(* IEC 61131-3 sources: CodesysTest/alpha/export/FBs, 6 files *)

(* ---- FB_CylinderLeak.pou.st ---- *)
(*#-#-#-#-#-#-#-#-#-#---Declaration---#-#-#-#-#-#-#-#-#-#-#-#-#*)

FUNCTION_BLOCK FB_CylinderLeak EXTENDS FB_PredictiveMaint
VAR_INPUT
	iExtended : BOOL;
	iRetracted : BOOL;
	maximumStrokeTime : REAL;
END_VAR
VAR_OUTPUT
	strokeTime : REAL;
END_VAR
VAR
	strokeTimer : TON := (PT := T#1H);
	extendedONS : R_TRIG;
	retractedONS : R_TRIG;
END_VAR
(*#-#-#-#-#-#-#-#-#-#---Implementation---#-#-#-#-#-#-#-#-#-#-#-#-#*)

extendedONS(CLK := iExtended);
retractedONS(CLK := iRetracted);

IF extendedONS.Q OR retractedONS.Q THEN
	strokeTime := TO_REAL(strokeTimer.ET) / 1000;
END_IF

strokeTimer(IN := NOT iExtended AND NOT iRetracted);

(* ---- FB_DriveTemp.pou.st ---- *)
(*#-#-#-#-#-#-#-#-#-#---Declaration---#-#-#-#-#-#-#-#-#-#-#-#-#*)

FUNCTION_BLOCK FB_DriveTemp EXTENDS FB_PredictiveMaint
VAR_INPUT
	iDriveTemp : DINT;
	maxTemp : REAL;
END_VAR
VAR_OUTPUT
	DriveTemp : REAL;
END_VAR
VAR
END_VAR
(*#-#-#-#-#-#-#-#-#-#---Implementation---#-#-#-#-#-#-#-#-#-#-#-#-#*)

DriveTemp := TO_REAL(iDriveTemp) / 10.0;

(* ---- FB_Throughput.pou.st ---- *)
(*#-#-#-#-#-#-#-#-#-#---Declaration---#-#-#-#-#-#-#-#-#-#-#-#-#*)

FUNCTION_BLOCK FB_Throughput
VAR_INPUT
	inCycle : BOOL;
	runtimeTimeout : REAL := 5.0;
	reset : BOOL;
END_VAR
VAR_OUTPUT
	BPM : REAL;
	BPMCycles : UDINT;
	BPMSeconds : UDINT;
	BPMIndication : STRING;
END_VAR
VAR
	resetRuntime : BOOL;
	resetRuntimeTimer : TON := (PT := T#0S);
	runtimeTimeoutTimer : Standard.TON;
	runtimeTimer : Standard.TON;
	actualRuntimeTimer : Standard.TON;
	timeoutONS : FB_ONS;
	inCycleONS : FB_ONS;
	runtimeSeconds : UDINT;
	runtimeMinutes : UDINT;
	runtimeHours : UDINT;
	runtimeDays : UDINT;
	runtimeSubtractedToGetFiveSeconds : UDINT;
	cycleStarted : BOOL;
	totalTempH : UDINT;
	totalTempM : UDINT;
	totalTempS : UDINT;
END_VAR
(*#-#-#-#-#-#-#-#-#-#---Implementation---#-#-#-#-#-#-#-#-#-#-#-#-#*)

// Runtime calculation. The goal is to capture actual runtime of the machine (i.e being used, including loading time)
inCycleONS(CLK := inCycle);
// Reset timeout time
IF inCycleONS.OSR THEN
	resetRuntime := TRUE;
	cycleStarted := TRUE;
	BPMCycles := BPMCycles + 1;
END_IF;

// After timeout, assume machine in unmanned
runtimeTimeoutTimer(IN := NOT resetRuntime, PT := TO_TIME(runtimeTimeout * 1000.0));
resetRuntime := FALSE;
timeoutONS(CLK := runtimeTimeoutTimer.Q);

// 1 second ticker while being used.
actualRuntimeTimer(IN := cycleStarted AND NOT actualRuntimeTimer.Q AND NOT runtimeTimeoutTimer.Q, PT := T#1S);

IF actualRuntimeTimer.Q THEN
	BPMSeconds := BPMSeconds + 1;
END_IF;

// Subtract 5 seconds after machine is abandoned
runtimeSubtractedToGetFiveSeconds := ANY_TO_UDINT(ABS(5.0 - runtimeTimeout));

IF timeoutONS.OSR THEN
	IF BPMSeconds > runtimeSubtractedToGetFiveSeconds THEN
		BPMSeconds := BPMSeconds - runtimeSubtractedToGetFiveSeconds;
	END_IF;
	cycleStarted := FALSE;
END_IF;

IF reset THEN
	BPMSeconds := 0;
	BPMCycles := 0;
END_IF;

// Concat to string for display
runtimeHours := BPMSeconds / 3600;
runtimeMinutes := (BPMSeconds MOD 3600) / 60;
runtimeSeconds := BPMSeconds MOD 60;

IF BPMSeconds <> 0 THEN
	BPM := ANY_TO_REAL(BPMCycles) / (ANY_TO_REAL(BPMSeconds) / 60.0);
ELSE
	BPM := 0.0;
END_IF;
BPMIndication := '';
BPMIndication := ANY_TO_STRING(runtimeHours);
BPMIndication := INSERT(BPMIndication, 'H  ', LEN(BPMIndication) + 2);
BPMIndication := INSERT(BPMIndication, ANY_TO_STRING(runtimeMinutes), LEN(BPMIndication));
BPMIndication := INSERT(BPMIndication, 'M ', LEN(BPMIndication));
BPMIndication := INSERT(BPMIndication, ANY_TO_STRING(runtimeSeconds), LEN(BPMIndication));
BPMIndication := INSERT(BPMIndication, 'S', LEN(BPMIndication));

(* ---- FB_WriteToFile.pou.st ---- *)
(*#-#-#-#-#-#-#-#-#-#---Declaration---#-#-#-#-#-#-#-#-#-#-#-#-#*)

FUNCTION_BLOCK FB_WriteToFile
VAR_INPUT
   xFilePath: STRING;
   xText_Write: STRING(5000);
   xAppend_OverWrite: BOOL;
   xAppend_Pos: UDINT;
   xWrite: BOOL;
   xRead: BOOL;
   xLine_No_To_Read: UDINT;
END_VAR
VAR_OUTPUT
   xText_Read: STRING(5000);
   xDone: BOOL;
END_VAR
VAR

// Write Variables
   xWrite_Trig: R_TRIG;
   xStart_Write: BOOL;
   xNew_Line: STRING(5000);

// Read Variables
   xRead_Trig: R_TRIG;
   xStart_Read: BOOL;
   xLine_Read: UDINT;

   hFile           : SysFile.RTS_IEC_HANDLE := SysFile.HandleConstants.RTS_INVALID_HANDLE;
   udiBytesRead    : LWORD;
   udiBytesCopied   : UDINT;
   udiWrite      : LWORD;
   udiFileSize     : UDINT;
   udiPos         : UDINT;

//(* Error Codes *)
   udiPosError          : SysFile.RTS_IEC_RESULT;
   udiCopyError      : SysFile.RTS_IEC_RESULT;
   udiDeleteError1      : SysFile.RTS_IEC_RESULT;
   udiDeleteError2      : SysFile.RTS_IEC_RESULT;
   udiWriteError1      : SysFile.RTS_IEC_RESULT;
   udiWriteError2      : SysFile.RTS_IEC_RESULT;
   udiWriteError3      : SysFile.RTS_IEC_RESULT;
   udiOpenError1      : SysFile.RTS_IEC_RESULT;
   udiOpenError2      : SysFile.RTS_IEC_RESULT;
   udiOpenError3      : SysFile.RTS_IEC_RESULT;
   udiOpenError4      : SysFile.RTS_IEC_RESULT;

   udiReadError1   : SysFile.RTS_IEC_RESULT;
   udiReadError2   : SysFile.RTS_IEC_RESULT;
   udiReadError3   : SysFile.RTS_IEC_RESULT;
   udiCloseError1   : SysFile.RTS_IEC_RESULT;
   udiCloseError2   : SysFile.RTS_IEC_RESULT;
   udiCloseError3   : SysFile.RTS_IEC_RESULT;
   udiCloseError4   : SysFile.RTS_IEC_RESULT;
   udiSizeError : SysFile.RTS_IEC_RESULT;
   udiDirDeleteError: UDINT;
   udiCreateError: UDINT;
END_VAR(*#-#-#-#-#-#-#-#-#-#---Implementation---#-#-#-#-#-#-#-#-#-#-#-#-#*)

xWrite_Trig();
//xWrite_Trig.PT:= T#500MS;
xWrite_Trig.CLK:= xWrite;
xStart_Write:= xWrite_Trig.Q;

xRead_Trig();
//xRead_Trig.PT:= T#500MS;
xRead_Trig.CLK:= xRead;
xStart_Read:= xRead_Trig.Q;

IF xStart_Write THEN
   xDone:= FALSE;
   IF xAppend_OverWrite THEN
   hFile:= SysFileOpen(szFile:= xFilePath, am:= ACCESS_MODE.AM_APPEND, pResult:= ADR(udiOpenError1));
   END_IF
   IF xAppend_OverWrite = FALSE THEN
      hFile:= SysFileOpen(szFile:= xFilePath, am:= ACCESS_MODE.AM_WRITE_PLUS, pResult:= ADR(udiOpenError1));
   END_IF
   udiPosError:= SysFileGetPos(hFile:= hFile, pulPos:= ADR(udiPos));
   IF hFile <> SysFile.HandleConstants.RTS_INVALID_HANDLE THEN
      xNew_Line:= concat('$n', xText_Write);
      IF udiPos = 16#0 THEN
         udiWrite:= SysFileWrite(hFile:= hFile, pbyBuffer:= ADR(xText_Write), ulSize:= INT_TO_UDINT(LEN(xText_Write)), pResult:= ADR(udiWriteError1));
      ELSE
         udiWrite:= SysFileWrite(hFile:= hFile, pbyBuffer:= ADR(xNew_Line), ulSize:= INT_TO_UDINT(LEN(xNew_Line)), pResult:= ADR(udiWriteError1));
      END_IF
      udiCloseError1:= SysFileClose(hFile:= hFile);
   END_IF
   xDone:= TRUE;
END_IF

IF xStart_Read THEN
   xDone:= FALSE;
   hFile:= SysFileOpen(szFile:= xFilePath, am:= ACCESS_MODE.AM_READ, pResult:= ADR(udiOpenError1));
   IF hFile <> SysFile.HandleConstants.RTS_INVALID_HANDLE THEN
      udiBytesRead := SysFileRead(hFile:= hFile, pbyBuffer:= ADR(xText_Read), ulSize:=SIZEOF(xText_Read), pResult:=ADR(udiReadError1));
      xText_Read[udiBytesRead]:= 0;
   END_IF
   //xDone:= TRUE;
END_IF

(* ---- GetTime.pou.st ---- *)
(*#-#-#-#-#-#-#-#-#-#---Declaration---#-#-#-#-#-#-#-#-#-#-#-#-#*)

FUNCTION_BLOCK GetTime
VAR_INPUT
END_VAR
VAR_OUTPUT
    currentDateAndTime : DATE_AND_TIME;

END_VAR
VAR
    iState                    : INT;
    udiUtcTime             : UDINT;
    udiUtcTimeLocal     : UDINT;
    strTimeDate         : SYSTIMEDATE;
    strTimeDateLocal     : SYSTIMEDATE;
    dtDateTimeUTC        : DATE_AND_TIME;
    timeLeftTime        : TIME;
    timeLeftDWORD        : DWORD;
    dDateUTC            : DATE;
    todTimeOfDayUTC        : TOD;

    tSysStartTime        : TIME;
    systimeStartNano    : SYSTIME;
    udiStartTimeResult    : UDINT;

    udiResult             : UDINT;

    GetDateAndTime            : DTU.GetDateAndTime;
    SetTimeZoneInformation    : DTU.SetTimeZoneInformation;

    dtCurrent                : DATE_AND_TIME;
    dtConcated                : DATE_AND_TIME;
    eWeekday                 : RTCLK.WEEKDAY;
    uiYear                     : UINT;
    uiMonth                     : UINT;
    uiDay                     : UINT;
    uiHour                     : UINT;
    uiMinute                 : UINT;
    uiSecond                 : UINT;

    dtuError                : DTU.ERROR;
END_VAR
(*#-#-#-#-#-#-#-#-#-#---Implementation---#-#-#-#-#-#-#-#-#-#-#-#-#*)

CASE iState OF

    0:
        iState:= 1;

    1:  // retrieves the target date and time, including the timezone information which was set before
        GetDateAndTime( xExecute:= TRUE);
        IF GetDateAndTime.xDone THEN
            dtCurrent:= GetDateAndTime.dtDateAndTime;
            GetDateAndTime(xExecute:= FALSE);
			currentDateAndTime := dtCurrent;
            //timeLeft := TIME_TO_DT(DT_TO_TIME(targetDate) - DT_TO_TIME(dttarget));
            iState:= 2;
        END_IF
        IF GetDateAndTime.xError THEN
            GetDateAndTime(xExecute:= FALSE);
            iState:= 32767;
        END_IF

    2: (*set a spedific date and time --> returns a variable of type DATE_AND_TIME
         DateConcat --> set only date information --> returns a variable of type DATE
         TODConcat  --> set only the time information  --> returns a variable of TOD (Time of day) *)
        IF dtuError = 0 THEN
            iState := 3;
        ELSE
            iState := 32767;
        END_IF

    3:  (*a DATE_AND_TIME variable is splitted in its parts, like year, month, day etc.
            DateSplit --> the same function for a DATE variable
            TODSplit  --> the same function for a TOD variable *)

        IF dtuError = 0 THEN
            iState:= 1;
        ELSE
            iState:= 32767;
        END_IF

    32767: ; //error

END_CASE

(* ---- SerialMotorTestFB.pou.st ---- *)
(*#-#-#-#-#-#-#-#-#-#---Declaration---#-#-#-#-#-#-#-#-#-#-#-#-#*)

FUNCTION_BLOCK SerialMotorTestFB
VAR_INPUT
    runMotorPB : BOOL;
END_VAR
VAR_OUTPUT
END_VAR
VAR
    //testMotor : FB_AppliedMotionStepServoRTU();
    //orientalMotor : FB_OrientalAZDrive();
END_VAR
(*#-#-#-#-#-#-#-#-#-#---Implementation---#-#-#-#-#-#-#-#-#-#-#-#-#*)

(*
orientalMotor(modbusInBuffer := OrientalMotorModbusRead,
                stepsPerInchSetpoint := 2122,
                reversePolarity := FALSE,
                operatingCurrentDefault := 100,
                modbusCommandOutBuffer := OrientalMotorCommandWrites,
                modbusParametersOutBuffer := OrientalMotorParameterWrites,
                triggerCommandWrite => OrientalMotorTriggerCommandWrite,
                triggerParameterWrite => OrientalMotorTriggerParameterWrite);
orientalMotor.Execute();
*)

IF runMotorPB THEN
    //testMotor.MoveDistance(12,100,100,215);
    //testMotor.HomeNow();

    //orientalMotor.MoveDistance(12,10000,10000,10000);
    runMotorPB := FALSE;
END_IF
